{attribute 'GeneratedUsingTerminal: EK1122-0000-0018'}
{attribute addProperty BoxType "EK1122-0000-0018"}
{attribute addProperty Id "Beckhoff_EL2xxxsub_EK1100EK1100_AB5A94672"}
{attribute addProperty CRC "2020924303"}
{attribute addProperty Size "2"}
TYPE Beckhoff_EL2xxxEK1122_7874DB8F EXTENDS EK1122_AB5A9467 :
STRUCT
	{attribute addProperty Name "Beckhoff_EL2xxxsub_EK1100"}
	{attribute addProperty PreviousPort "Beckhoff EL2xxxEK1122 : D"}
	Beckhoff_EL2xxxsub_EK1100 : EK1100_AB5A9467;
END_STRUCT
END_TYPE

(* stored: Version 1.2.0.0, ProductVersion 3.1.4024.9
   DUT Beckhoff_EL2xxxEK1122_7874DB8F: Id {03275dab-6f0d-4d52-9c75-719f11ea3fb6} *)
